(* IEC 61131-3 sources: Std_PalletMover/Class/MainLiftControl, 1 file *)

(* ---- MainLiftControl.st ---- *)
(*!
<Class
	Name               = "MainLiftControl"
	Revision           = "0.0"
	RealtimeTask       = "false"
	CyclicTask         = "false"
	BackgroundTask     = "false"
	Sigmatek           = "false"
	OSInterface        = "false"
	HighPriority       = "false"
	Automatic          = "false"
	UpdateMode         = "Prescan"
	SharedCommandTable = "true"
	Objectsize         = "(660,180)">
	<Channels>
		<Server Name="ActualHeight" Visualized="false" Initialize="false" WriteProtected="true" Retentive="false"/>
		<Server Name="SetHeight" Visualized="false" Initialize="false" WriteProtected="true" Retentive="false"/>
		<Server Name="SetSpeed" Visualized="false" Initialize="false" WriteProtected="true" Retentive="false"/>
		<Server Name="State" Visualized="false" Initialize="false" WriteProtected="true" Retentive="false"/>
		<Client Name="_LMCAxis" Required="true" Internal="true"/>
		<Client Name="ActuValveDown" Required="true" Internal="false"/>
		<Client Name="ActuValveUp" Required="true" Internal="false"/>
		<Client Name="AgvConfig" Required="true" Internal="false"/>
		<Client Name="AgvSettings" Required="true" Internal="false"/>
		<Client Name="Ain_AnalogPosition" Required="true" Internal="false"/>
		<Client Name="HydroController" Required="true" Internal="true"/>
		<Client Name="I_Lift" Required="true" Internal="true"/>
		<Client Name="SensorMaxHeight" Required="false" Internal="false"/>
		<Client Name="SensorMinHeight" Required="true" Internal="false"/>
		<Client Name="Speed" Required="true" Internal="false"/>
	</Channels>
	<Network Name="MainLiftControl">
		<!-- List of Components in this network -->
		<Components>
			<Object
				Name       = "_base"
				Class      = "PeripheralsBase"
				Position   = "(218,120)"
				Visualized = "false">
				<Channels>
					<Server Name="ObjectStatus"/>
					<Server Name="ToObject"/>
					<Client Name="op_LogData"/>
					<Client Name="p_NextObject"/>
				</Channels>
			</Object>
			<Object
				Name           = "_LMCAxis"
				Class          = "_LMCAxis"
				Position       = "(1080,870)"
				Visualized     = "true"
				Remotely       = "true"
				RealTime       = "1 ms"
				CyclicTime     = "10 ms"
				BackgroundTime = "100 ms">
				<Channels>
					<Server Name="AbsEncoder"/>
					<Server Name="ActPos"/>
					<Server Name="ActVelocity"/>
					<Server Name="AEmergency" Value="0"/>
					<Server Name="AMax" Value="50m"/>
					<Server Name="AxisError"/>
					<Server Name="AxisStatus"/>
					<Server Name="Control"/>
					<Server Name="Destination"/>
					<Server Name="ErrorConfig" Value="2#0000000001000000"/>
					<Server Name="ExUnits" Value="65536"/>
					<Server Name="IntUnits" Value="100mm"/>
					<Server Name="JMax" Value="0"/>
					<Server Name="Modulo" Value="0"/>
					<Server Name="MoveType" Value="_RAMP_Profile"/>
					<Server Name="Override"/>
					<Server Name="PosMode"/>
					<Server Name="Resolution" Value="1"/>
					<Server Name="SetPos"/>
					<Server Name="SetVelocity"/>
					<Server Name="SimulateMode" Value="0"/>
					<Server Name="SWMaxPos" Value="0"/>
					<Server Name="SWMinPos" Value="0"/>
					<Server Name="Tjerk" Value="0"/>
					<Server Name="VMax" Value="5m"/>
					<Client Name="ActPosition"/>
					<Client Name="Config" Value="0"/>
					<Client Name="Emergency"/>
					<Client Name="HWError"/>
					<Client Name="HWMax"/>
					<Client Name="HWMin"/>
					<Client Name="HWReady"/>
					<Client Name="ID" Value="0"/>
					<Client Name="LatchPos"/>
					<Client Name="LMCController"/>
					<Client Name="LMCPostRtWorkTrigger"/>
					<Client Name="LMCPreRtWorkTrigger"/>
					<Client Name="Provider"/>
					<Client Name="RefSwitch"/>
					<Client Name="ZImpulse"/>
				</Channels>
			</Object>
			<Object
				Name       = "HydroController"
				Class      = "HydroController"
				Position   = "(510,930)"
				Visualized = "true"
				Remotely   = "true">
				<Channels>
					<Server Name="Signal_Input"/>
					<Server Name="XW"/>
					<Server Name="XwMax"/>
					<Client Name="cDraglimit" Value="0"/>
					<Client Name="cEmerStop"/>
					<Client Name="cImode"/>
					<Client Name="cMaxSignal1" Value="40"/>
					<Client Name="cMaxSignal2" Value="40"/>
					<Client Name="cMaxSpeed" Value="100"/>
					<Client Name="cOffSignal" Value="20"/>
					<Client Name="HWErrorQuit"/>
					<Client Name="iHWErrors"/>
					<Client Name="oActive"/>
					<Client Name="odirection"/>
					<Client Name="oOutputSignal"/>
					<Client Name="vHWDelay"/>
					<Client Name="vKD1"/>
					<Client Name="vKD2"/>
					<Client Name="vKI1"/>
					<Client Name="vKI2"/>
					<Client Name="vKV1"/>
					<Client Name="vKV2"/>
					<Client Name="vVU1" Value="45"/>
					<Client Name="vVU2" Value="45"/>
				</Channels>
			</Object>
			<Object
				Name       = "I_Lift"
				Class      = "I_Lift"
				Position   = "(510,360)"
				Visualized = "false">
				<Channels>
					<Server Name="ActualHeight"/>
					<Server Name="ClassSvr"/>
					<Server Name="SetHeight"/>
					<Server Name="SetSpeed"/>
					<Server Name="State"/>
				</Channels>
			</Object>
		</Components>
		<Comments>
		</Comments>
		<!-- List of Connections in this network -->
		<Connections>
			<Connection Source="this.ToObject" Destination="_base.ToObject" Vertices="(1918,210),(804,210),"/>
			<Connection Source="_base.op_LogData" Destination="this.op_LogData" Vertices="(218,210),(38,210),"/>
			<Connection Source="_base.p_NextObject" Destination="this.p_NextObject" Vertices="(218,270),(38,270),"/>
			<Connection Source="this.I_Lift" Destination="I_Lift.ClassSvr"/>
			<Connection Source="this._LMCAxis" Destination="_LMCAxis.Control"/>
			<Connection Source="this.HydroController" Destination="HydroController.Signal_Input"/>
			<Connection Source="_LMCAxis.LMCController" Destination="HydroController.Signal_Input" Vertices="(1080,1020),(948,1020),"/>
			<Connection Source="this.ActualHeight" Destination="I_Lift.ActualHeight" Vertices="(1918,330),(1156,510),"/>
			<Connection Source="this.SetHeight" Destination="I_Lift.SetHeight" Vertices="(1918,390),(1156,570),"/>
			<Connection Source="this.SetSpeed" Destination="I_Lift.SetSpeed" Vertices="(1918,450),(1156,630),"/>
			<Connection Source="this.State" Destination="I_Lift.State" Vertices="(1918,510),(1156,690),"/>
		</Connections>
		<!-- Headerfiles -->
		<Options>
		</Options>
	</Network>
</Class>
*)
#pragma using PeripheralsBase

MainLiftControl : CLASS
: PeripheralsBase
  //Servers:
	ActualHeight 	: SvrCh_DINT;
	SetHeight 	: SvrCh_DINT;
	SetSpeed 	: SvrCh_DINT;
	State 	: SvrCh_LiftState_PTofCls_I_Lift;
  //Clients:
	I_Lift 	: CltChCmd_I_Lift;
	AgvConfig 	: CltChCmd_AgvConfig;
	AgvSettings 	: CltCh_DINT;
	Ain_AnalogPosition 	: CltCh_DINT;
	SensorMaxHeight 	: CltCh_DINT;
	SensorMinHeight 	: CltCh_DINT;
	ActuValveUp 	: CltCh_DINT;
	ActuValveDown 	: CltCh_DINT;
	Speed 	: CltCh_DINT;
	HydroController 	: CltChCmd_HydroController;
	_LMCAxis 	: CltChCmd__LMCAxis;
  //Variables:
		ConnectionMaxHeightSensor 	: ^CHAR;
		Stepper 	: DINT;
  //Functions:

	FUNCTION VIRTUAL GLOBAL HandleOperational
		VAR_OUTPUT
			RetValue 	: DINT;
		END_VAR;

	FUNCTION VIRTUAL GLOBAL Handleconfiguration
		VAR_OUTPUT
			RetValue 	: DINT;
		END_VAR;

	FUNCTION VIRTUAL GLOBAL HandleGetSettings
		VAR_OUTPUT
			RetValue 	: DINT;
		END_VAR;

	FUNCTION GetConfigSettings;

	FUNCTION GetSettings;

	FUNCTION VIRTUAL GLOBAL ActualHeight::Read
		VAR_OUTPUT
			output (EAX) 	: DINT;
		END_VAR;

	FUNCTION VIRTUAL GLOBAL SetHeight::Read
		VAR_OUTPUT
			output (EAX) 	: DINT;
		END_VAR;

	FUNCTION VIRTUAL GLOBAL SetSpeed::Read
		VAR_OUTPUT
			output (EAX) 	: DINT;
		END_VAR;

	FUNCTION VIRTUAL GLOBAL State::Read
		VAR_OUTPUT
			output (EAX) 	: I_Lift::LiftState;
		END_VAR;
  //Tables:
	FUNCTION @STD
		VAR_OUTPUT
			ret_code	: CONFSTATES;
		END_VAR;
	FUNCTION GLOBAL TAB @CT_;
END_CLASS;

#pragma using _LMCAxis
#pragma using HydroController
#pragma using I_Lift
#pragma usingLtd AgvConfig

FUNCTION VIRTUAL GLOBAL MainLiftControl::ActualHeight::Read
	VAR_OUTPUT
		output (EAX) 	: DINT;
	END_VAR

	ActualHeight := I_Lift.ActualHeight.Read();
	output := ActualHeight;

END_FUNCTION

FUNCTION VIRTUAL GLOBAL MainLiftControl::SetHeight::Read
	VAR_OUTPUT
		output (EAX) 	: DINT;
	END_VAR

	SetHeight := I_Lift.SetHeight.Read();
	output := SetHeight;

END_FUNCTION

FUNCTION VIRTUAL GLOBAL MainLiftControl::SetSpeed::Read
	VAR_OUTPUT
		output (EAX) 	: DINT;
	END_VAR

	SetSpeed := I_Lift.SetSpeed.Read();
	output := SetSpeed;

END_FUNCTION

FUNCTION VIRTUAL GLOBAL MainLiftControl::State::Read
	VAR_OUTPUT
		output (EAX) 	: I_Lift::LiftState;
	END_VAR

	State := I_Lift.State.Read();
	output := State;

END_FUNCTION

FUNCTION VIRTUAL GLOBAL MainLiftControl::HandleOperational
	VAR_OUTPUT
		RetValue 	: DINT;
	END_VAR

END_FUNCTION

FUNCTION VIRTUAL GLOBAL MainLiftControl::Handleconfiguration
	VAR_OUTPUT
		RetValue 	: DINT;
	END_VAR

    RetValue := False;;

    case Stepper of

        0:
                 GetConfigSettings();
                Stepper += 1;
        1:
              SensorMaxHeight := SensorMaxHeight.Read();

                // RetValue := true;
      end_case;

END_FUNCTION

FUNCTION VIRTUAL GLOBAL MainLiftControl::HandleGetSettings
	VAR_OUTPUT
		RetValue 	: DINT;
	END_VAR

END_FUNCTION

FUNCTION MainLiftControl::GetConfigSettings

// Use sensor and make connection with hardware

// Get config
ConnectionMaxHeightSensor := AgvConfig.GetStringValue(Path:="AGV.Peripherals.BasicActuator.Connection.SensorMaxHeight");

// Set connection's
if ConnectionMaxHeightSensor<> nil then
   ConnectClientChannels(ConnectionMaxHeightSensor);
end_if;

END_FUNCTION

FUNCTION MainLiftControl::GetSettings

END_FUNCTION
